TYPE ST_FSoE_04Byte :
STRUCT
	CMD		: BYTE;
	SafeData1 	: WORD;
	CRC1		: WORD;
	SafeData2 	: WORD;
	CRC2		: WORD;
	ConnID		: WORD;
END_STRUCT
END_TYPE

(* stored: Version 1.1.0.1, ProductVersion 3.1.4024.5
   DUT ST_FSoE_04Byte: Id {86095c8f-9fad-41a5-9fa2-dfd9d8668843} *)
